{attribute 'qualified_only'}
{attribute 'strict'}
{attribute 'to_string'}
TYPE EBaudrate :
(
	_9600   := 6,
	_19200  := 7,
	_38400  := 8,
	_57600  := 9,
	_115200 := 10
);
END_TYPE

(* stored: Version 1.1.0.1, ProductVersion 3.1.4024.12
   DUT EBaudrate: Id {78de0957-d592-472b-8483-6b4260cc731e} *)
